// Mitsubishi GX Works2 project: 전철제어기   PLC: Q03UDV

PROGRAM MAIN
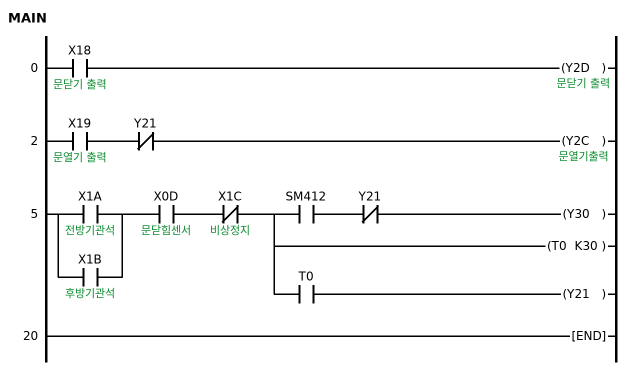
0     LD      X18  ; 문닫기 출력
      OUT     Y2D  ; 문닫기 출력
2     LD      X19  ; 문열기 출력
      ANI     Y21
      OUT     Y2C  ; 문열기출력
5     LD      X1A  ; 전방기관석
      OR      X1B  ; 후방기관석
      AND     X0D  ; 문닫힘센서
      ANI     X1C  ; 비상정지
      MPS
      AND     SM412
      ANI     Y21
      OUT     Y30
      MPP
      OUT     T0 K30
      AND     T0
      OUT     Y21
20    END
END_PROGRAM
